FUNCTION_BLOCK PML_StatePattern_Base
VAR_INPUT
END_VAR
VAR_OUTPUT
END_VAR
VAR
	stateMachine : PMLStateMachine;
	iStateMachine : IPmlStateMachine := stateMachine;
	undefined : Undefined_State(THIS, iStateMachine);
	aborting : Aborting_State(THIS, iStateMachine);
	aborted : Aborted_State(THIS, iStateMachine);
	clearing : Clearing_State(THIS, iStateMachine);
	stopped : Stopped_State(THIS, iStateMachine);
	resetting : Resetting_State(THIS, iStateMachine);
	idle : Idle_State(THIS, iStateMachine);
	starting : Starting_State(THIS, iStateMachine);
	execute : Execute_State(THIS, iStateMachine);
	iState : ITF_State := undefined;
END_VAR

iState.Cycle();
stateMachine();

METHOD SetState : BOOL
VAR_INPUT
  newState : ITF_State;
END_VAR
THIS^.iState := newState;
END_METHOD

END_FUNCTION_BLOCK

(* stored: Version 1.1.0.1, ProductVersion 3.1.4024.12
   POU PML_StatePattern_Base: Id {ba6afb7a-8005-4e25-84a5-74a3195b2390}, SpecialFunc None
   Method SetState: Id {dfdcdd31-ba2b-4b00-9c72-539badf1770b} *)
